# EPICS substitutions: vaccelApp/Db/transfer.substitutions
file db/transfer_function.rec
{
	pattern{ ELEMENT,   HW2PHYS               }
               { q1m1d1r,   1.1270572620311009e-02}
               { q1m1d2r,   1.1270572620311009e-02}
               { q1m1d3r,   1.1270572620311009e-02}
               { q1m1d4r,   1.1270572620311009e-02}
               { q1m1d5r,   1.1270572620311009e-02}
               { q1m1d6r,   1.1270572620311009e-02}
               { q1m1d7r,   1.1270572620311009e-02}
               { q1m1d8r,   1.1270572620311009e-02}

               { q1m1t1r,   1.1270572620311009e-02}
               { q1m1t2r,   1.1270572620311009e-02}
               { q1m1t3r,   1.1270572620311009e-02}
               { q1m1t4r,   1.1270572620311009e-02}
               { q1m1t5r,   1.1270572620311009e-02}
               { q1m1t6r,   1.1270572620311009e-02}
               { q1m1t7r,   1.1270572620311009e-02}
               { q1m1t8r,   1.1270572620311009e-02}
}
